Fanuc KAREL source: kb00196.KL

-- PROVISIONAL review KL for V770-1; original PC SHA256 cff6cb61db22f7dcce2385c104708873171f8fab404fca9b7a325b0d12c4a964
-- Incomplete behavior may be omitted. Consult companion uncertainty JSON. Do not deploy.
PROGRAM KB00196
%NOLOCKGROUP
BEGIN
  -- UNRESOLVED_PC offsets 5-14; opcodes 3F,75
  -- UNRESOLVED_PC offsets 19-26; opcodes 9D,23
  -- UNRESOLVED_PC offsets 31-38; opcodes 9D,23
  -- UNRESOLVED_PC offsets 43-52; opcodes 3F,75
  -- UNRESOLVED_PC offsets 57-89; opcodes 27,22,2A,22,22,22,2A,31
  -- UNRESOLVED_PC offsets 94-98; opcodes 7F
END KB00196
